// TIA Portal V19 export
DATA_BLOCK "FLUSH DB"   // DB41
{ S7_Optimized_Access := 'TRUE' }
// stored: MemoryReserve 100
   VAR
      "ABFV 101 MULTIGRADE FILTER VALVE" : Bool;
      "ABFV 102 MULTIGRADE FILTER VALVE" : Bool;
      "ABFV 103 MULTIGRADE FILTER VALVE" : Bool;
      "ABFV 104 MULTIGRADE FILTER VALVE" : Bool;
      "ABFV 105 MULTIGRADE FILTER VALVE" : Bool;
      "ABV 201 UF VALVE" : Bool;
      "ABFV 201 UF VALVE" : Bool;
      "ABFV 202 UF VALVE" : Bool;
      "ABFV 203 UF VALVE" : Bool;
      "ABFV 204 UF VALVE" : Bool;
      "ABFV 205 UF VALVE" : Bool;
      "ABFV 206 UF VALVE" : Bool;
      "ABFV 207 UF VALVE" : Bool;
      "ABFV 208 UF VALVE" : Bool;
      "ABFV 101 MULTIGRADE FILTER VALVE_CLOSE" : Bool;
      "ABFV 102 MULTIGRADE FILTER VALVE_CLOSE" : Bool;
      "ABFV 103 MULTIGRADE FILTER VALVE_CLOSE" : Bool;
      "ABFV 104 MULTIGRADE FILTER VALVE_CLOSE" : Bool;
      "ABFV 105 MULTIGRADE FILTER VALVE_CLOSE" : Bool;
      "ABV 201 UF VALVE_CLOSE" : Bool;
      "ABFV 201 UF VALVE_CLOSE" : Bool;
      "ABFV 202 UF VALVE_CLOSE" : Bool;
      "ABFV 203 UF VALVE_CLOSE" : Bool;
      "ABFV 204 UF VALVE_CLOSE" : Bool;
      "ABFV 205 UF VALVE_CLOSE" : Bool;
      "ABFV 206 UF VALVE_CLOSE" : Bool;
      "ABFV 207 UF VALVE_CLOSE" : Bool;
      "ABFV 208 UF VALVE_CLOSE" : Bool;
   END_VAR
BEGIN
END_DATA_BLOCK
